(* PLC project 117_1_V0.5.project, CODESYS CODESYS V3.5 SP17 Patch 3 *)
(* stored: creationDateTime 1970-01-01T00:00:00, modificationDateTime 2026-03-26T18:14:32.4070562 *)

FUNCTION_BLOCK SwitchingWithFeedbackControl
  VAR_INPUT
    xEnable : BOOL := FALSE;
    xInputSignal : BOOL := FALSE;
    xOutputSignal : BOOL := FALSE;
    waitTimeSwitch : TIME := TIME#2s0ms;
  END_VAR
  VAR
    WaitingTimer : WaitingTimer;
  END_VAR
  VAR_OUTPUT
    xForceOutputSignal : BOOL := FALSE;
    xSelfStatus : SW_STATUS := SW_STATUS.NONE;
  END_VAR

            // Если нет команды — ничего не делаем
IF NOT xEnable THEN
		WaitingTimer(xExecute := FALSE);
		xForceOutputSignal	:= FALSE;
		xSelfStatus			:= SW_STATUS.NONE;
    RETURN;
END_IF

// Если выход ещё не включён — включаем
IF NOT xOutputSignal THEN
    xForceOutputSignal := TRUE;
    RETURN;
END_IF

// Запуск таймера ожидания обратной связи
WaitingTimer(
    xExecute		:= TRUE,
    xCondition		:= xInputSignal,
    tWaitingTime	:= waitTimeSwitch);
	xSelfStatus := SW_STATUS.WAITING;

// Обратная связь получена
IF WaitingTimer.xDone THEN
    WaitingTimer(xExecute := FALSE);
    xSelfStatus	 := SW_STATUS.DONE;

// Таймаут
ELSIF WaitingTimer.xTimeOutError THEN
    WaitingTimer(xExecute := FALSE);
    xSelfStatus	 := SW_STATUS.TIMEOUT_ERROR;

END_IF


          
END_FUNCTION_BLOCK
